# EPICS autosave request: iocBoot/sioc-esb-pv04/pv.req
file ../pvCommon.req P=$(P)
file ../scanPv.req P=$(P)
